FUNCTION EXECUTE_FUNCTION : BOOL
VAR_INPUT
	FUNCT_NAME :STRING [255];
END_VAR
VAR
END_VAR

IF FUNCT_NAME = 'LOAD_FUKUDA' THEN
	//LOAD_FUKUDA(INPUT_VAR.I_CURRENT_TRANSACTION.STATION_NUMBER_LOAD,INPUT_VAR.I_CURRENT_TRANSACTION.JIG_INDEX_LOAD,INPUT_VAR.I_CURRENT_TRANSACTION.TRANSPORT_INDEX);
	INPUT_VAR.I_FUNC_CALLED:=TRUE;
	LOAD_FUKUDA();
END_IF
//INPUT_VAR.I_FUNCTION_NAME:='';

END_FUNCTION

(* stored: Version 1.1.0.1, ProductVersion 3.1.4020.12
   POU EXECUTE_FUNCTION: Id {51038094-f217-43fa-bbc0-fca0bb742f38}, SpecialFunc None *)
